# EPICS autosave request: iocBoot/iocCalc/auto_settings.req
file userCalcs10_settings.req P=$(P)
file userCalcN_settings.req P=$(P),N=I_Detector
file userTransforms10_settings.req P=$(P)
file userStringCalcs10_settings.req P=$(P)
file userAve10_settings.req P=$(P)
